Universal Robots PolyScope program: wrs2020_taskboard_belt_v2.urp

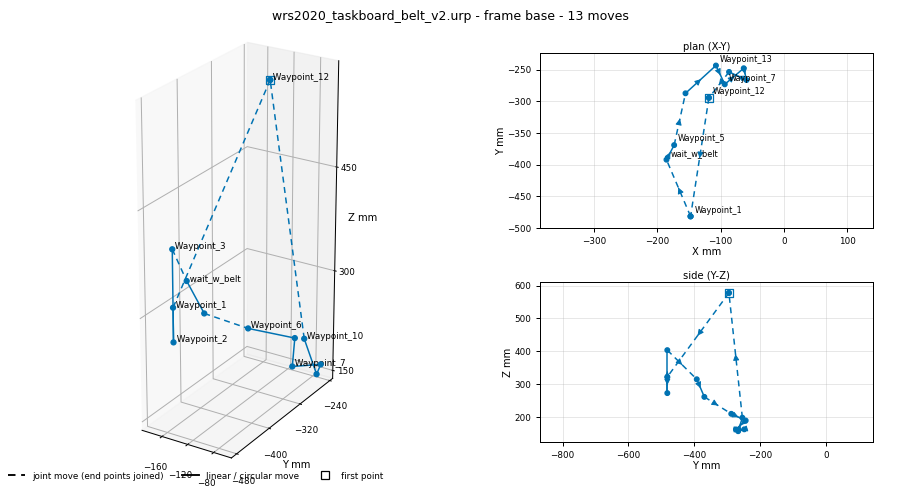
[picture p0: tool path of wrs2020_taskboard_belt_v2.urp in frame base, 13 of 13 moves have a stored position in this frame; points joined in program order, loops and branches not executed]
Program wrs2020_taskboard_belt_v2 (installation=default directory=/programs createdIn=5.6.0.90886 lastSavedIn=5.6.0.90886 robotSerialNumber=20205500180)
Calibrated DH parameters: a=[0.000135, -0.030981, -0.334292, 0.000083, 0.000088, 0]; d=[0.162656, 258.79096, -331.603246, 72.945842, 0.099724, 0.099562]; alpha=[1.569535, 0.001639, 0.002824, 1.569633, -1.569323, 0]; deltaTheta=[0, 1.497881, -2.049261, 0.551379, 0, 0]
Robot Program (runOnlyOnce=true)
  Set NoAction tcp=TCP
  MoveJ speed 60 deg/s, acceleration 80 deg/s^2 (useActiveTCP=false) tcp=TCP; feature=Base
    Waypoint Waypoint_12: TCP in base x=-118.553 y=-294.346 z=577.587 mm, rx=1.3176 ry=2.7241 rz=-0.2718 rad; joints [40.024, -118.444, 99.589, -78.038, -80.282, 2.128] deg
  URCap Gripper (Robotiq_Grippers, Robotiq Inc.) dataModel(position=48.23529411764706, force=100.0, speed=100.0, positionInDouble=48.23529411764706, forceInDouble=100.0, speedInDouble=100.0, slaveIds=[9], blocking=true)
  MoveJ speed 120 deg/s, acceleration 100 deg/s^2 (useActiveTCP=false) tcp=TCP; feature=Base
    Waypoint Waypoint_1: TCP in base x=-147.509 y=-481.576 z=322.425 mm, rx=-2.2532 ry=2.177 rz=0.038 rad; joints [57.916, -85.82, 110.34, -113.684, -91.081, -124] deg; TCP offset x=0 y=0 z=0 mm, rx=0 ry=0 rz=0 rad
    MoveL speed 50 mm/s, acceleration 1200 mm/s^2 (useActiveTCP=false) tcp=TCP; feature=Base
      Waypoint Waypoint_2: TCP in base x=-147.509 y=-481.576 z=273.212 mm, rx=2.2507 ry=-2.1796 rz=-0.0127 rad; joints [57.763, -82.536, 115.155, -122.915, -90.37, -124] deg; TCP offset x=0 y=0 z=0 mm, rx=0 ry=0 rz=0 rad
  URCap Gripper (Robotiq_Grippers, Robotiq Inc.) dataModel(position=100.0, force=100.0, speed=100.0, positionInDouble=100.0, forceInDouble=100.0, speedInDouble=100.0, slaveIds=[9], blocking=true)
  MoveL speed 250 mm/s, acceleration 1200 mm/s^2 (useActiveTCP=false) tcp=TCP; feature=Base
    Waypoint Waypoint_3: motionParameters(jointSpeed=1.047198 jointAcceleration=1.396263 cartesianSpeed=0.05 cartesianAcceleration=1.2); TCP in base x=-147.509 y=-481.576 z=403.735 mm, rx=2.2497 ry=-2.1806 rz=-0.0127 rad; joints [57.78, -89.668, 102.124, -102.752, -90.379, -124] deg; TCP offset x=0 y=0 z=0 mm, rx=0 ry=0 rz=0 rad
    MoveJ speed 60 deg/s, acceleration 80 deg/s^2 (useActiveTCP=false) tcp=TCP; feature=Base
      Waypoint wait_w_belt: TCP in base x=-185.572 y=-392.078 z=315.254 mm, rx=-1.4441 ry=1.9502 rz=-1.0486 rad; joints [37.028, -91.796, 114.934, -76.388, -46.414, -141.19] deg
  Popup Message (haltProgram=false message=wait for b_bot to move hook into belt (when b says 1) inputType=Text)
  MoveL speed 250 mm/s, acceleration 1200 mm/s^2 (useActiveTCP=false) tcp=TCP; feature=Base
    Waypoint Waypoint_5: TCP in base x=-173.43 y=-369.039 z=261.712 mm, rx=-1.282 ry=1.8047 rz=-1.1483 rad; joints [34.616, -88.409, 119.828, -68.558, -43.225, -150.47] deg
  MoveJ speed 60 deg/s, acceleration 80 deg/s^2 (useActiveTCP=false) tcp=TCP; feature=Base
    Waypoint Waypoint_6: TCP in base x=-155.523 y=-287.24 z=210.263 mm, rx=-1.031 ry=1.6203 rz=-1.5379 rad; joints [21.885, -87.537, 130.935, -50.465, -40.317, -177.586] deg
  MoveL speed 250 mm/s, acceleration 1200 mm/s^2 (useActiveTCP=false) tcp=TCP; feature=Base
    Waypoint Waypoint_13: TCP in base x=-107.458 y=-243.362 z=189.808 mm, rx=-0.909 ry=1.7261 rz=-1.6615 rad; joints [13.916, -96.788, 144.22, -53.106, -38.64, -178.723] deg
    Waypoint Waypoint_7: TCP in base x=-93.501 y=-273.032 z=162.831 mm, rx=-0.9044 ry=1.7298 rz=-1.6658 rad; joints [21.869, -90.172, 144.622, -61.38, -30.363, -177.16] deg
  Popup Message (haltProgram=false message=wait for b_bot to tension inputType=Text)
  MoveL speed 250 mm/s, acceleration 1200 mm/s^2 (useActiveTCP=false) tcp=TCP; feature=Base
    Waypoint Waypoint_8: TCP in base x=-63.539 y=-247.671 z=163.129 mm, rx=-0.7441 ry=1.8696 rz=-1.7976 rad; joints [15.11, -101.236, 153.772, -59.958, -25.437, -176.345] deg
  MoveL speed 250 mm/s, acceleration 1200 mm/s^2 (useActiveTCP=false) tcp=TCP; feature=Base
    Waypoint Waypoint_9: TCP in base x=-59.125 y=-266.29 z=157.434 mm, rx=-0.7441 ry=1.8696 rz=-1.7976 rad; joints [21.298, -97.571, 152.76, -64.841, -19.306, -173.924] deg
  Popup Message (haltProgram=false message=wait for b_bot to thread belt inputType=Text)
  URCap Gripper (Robotiq_Grippers, Robotiq Inc.) dataModel(position=80.3921568627451, force=0.0, speed=0.0, positionInDouble=80.3921568627451, forceInDouble=0.0, speedInDouble=0.0, slaveIds=[9], blocking=true)
  MoveL speed 250 mm/s, acceleration 1200 mm/s^2 (useActiveTCP=false) tcp=TCP; feature=Base
    Waypoint Waypoint_10: TCP in base x=-86.692 y=-253.478 z=198.507 mm, rx=-0.7729 ry=1.8477 rz=-1.7806 rad; joints [15.395, -103.398, 147.395, -51.019, -26.952, -177] deg; TCP offset x=0 y=0 z=0 mm, rx=0 ry=0 rz=0 rad
  MoveJ speed 60 deg/s, acceleration 80 deg/s^2 (useActiveTCP=false) tcp=TCP; feature=Base
    Waypoint Waypoint_11: TCP in base x=-118.553 y=-294.346 z=577.587 mm, rx=1.3176 ry=2.7241 rz=-0.2718 rad; joints [40.024, -118.444, 99.589, -78.038, -80.282, 2.128] deg
